(* IEC 61131-3 sources: RSI_PLC_Generation/artifacts/nas_qwen38_quantized_20260915/evidence/verification_20260915_132135, 1 file *)

(* ---- plc_smoke.st ---- *)
FUNCTION_BLOCK FB_StartStop
VAR_INPUT
    StartButton : BOOL;
    StopButton : BOOL;
END_VAR
VAR_OUTPUT
    Motor : BOOL;
END_VAR

IF StopButton THEN
    Motor := FALSE;
ELSIF StartButton THEN
    Motor := TRUE;
ELSE
    Motor := Motor;
END_IF;
END_FUNCTION_BLOCK
